# EPICS substitutions: iocBoot/ioczzz/zedLOreg6.substitutions
# base address 0x43c50000
file "$(TOP)/zzzApp/Db/zedLOreg.template"
{
pattern
{P,R,C,N, SCAN}
{zzz:,reg6_,6,0,8}
{zzz:,reg6_,6,1,8}
{zzz:,reg6_,6,2,8}
{zzz:,reg6_,6,3,8}
{zzz:,reg6_,6,4,8}
{zzz:,reg6_,6,5,8}
{zzz:,reg6_,6,6,8}
{zzz:,reg6_,6,7,8}
{zzz:,reg6_,6,8,8}
{zzz:,reg6_,6,9,8}
{zzz:,reg6_,6,10,8}
{zzz:,reg6_,6,11,8}
{zzz:,reg6_,6,12,8}
{zzz:,reg6_,6,13,8}
{zzz:,reg6_,6,14,8}
{zzz:,reg6_,6,15,8}
{zzz:,reg6_,6,16,8}
{zzz:,reg6_,6,17,8}
{zzz:,reg6_,6,18,8}
{zzz:,reg6_,6,19,8}
{zzz:,reg6_,6,20,8}
{zzz:,reg6_,6,21,8}
{zzz:,reg6_,6,22,8}
{zzz:,reg6_,6,23,8}
{zzz:,reg6_,6,24,8}
{zzz:,reg6_,6,25,8}
{zzz:,reg6_,6,26,8}
{zzz:,reg6_,6,27,8}
{zzz:,reg6_,6,28,8}
{zzz:,reg6_,6,29,8}

{zzz:,reg6_,6,30,8}
{zzz:,reg6_,6,31,8}
{zzz:,reg6_,6,32,8}
{zzz:,reg6_,6,33,8}
{zzz:,reg6_,6,34,8}
{zzz:,reg6_,6,35,8}
{zzz:,reg6_,6,36,8}
{zzz:,reg6_,6,37,8}
{zzz:,reg6_,6,38,8}
{zzz:,reg6_,6,39,8}

{zzz:,reg6_,6,40,8}
{zzz:,reg6_,6,41,8}
{zzz:,reg6_,6,42,8}
{zzz:,reg6_,6,43,8}
{zzz:,reg6_,6,44,8}
{zzz:,reg6_,6,45,8}
{zzz:,reg6_,6,46,8}
{zzz:,reg6_,6,47,8}
{zzz:,reg6_,6,48,8}
{zzz:,reg6_,6,49,8}

{zzz:,reg6_,6,50,8}
{zzz:,reg6_,6,51,8}
{zzz:,reg6_,6,52,8}
{zzz:,reg6_,6,53,8}
{zzz:,reg6_,6,54,8}
{zzz:,reg6_,6,55,8}
{zzz:,reg6_,6,56,8}
{zzz:,reg6_,6,57,8}
{zzz:,reg6_,6,58,8}
{zzz:,reg6_,6,59,8}

{zzz:,reg6_,6,60,8}
{zzz:,reg6_,6,61,8}
{zzz:,reg6_,6,62,8}
{zzz:,reg6_,6,63,8}
{zzz:,reg6_,6,64,8}
{zzz:,reg6_,6,65,8}
{zzz:,reg6_,6,66,8}
{zzz:,reg6_,6,67,8}
{zzz:,reg6_,6,68,8}
{zzz:,reg6_,6,69,8}

{zzz:,reg6_,6,70,8}
{zzz:,reg6_,6,71,8}
{zzz:,reg6_,6,72,8}
{zzz:,reg6_,6,73,8}
{zzz:,reg6_,6,74,8}
{zzz:,reg6_,6,75,8}
{zzz:,reg6_,6,76,8}
{zzz:,reg6_,6,77,8}
{zzz:,reg6_,6,78,8}
{zzz:,reg6_,6,79,8}

{zzz:,reg6_,6,80,8}
{zzz:,reg6_,6,81,8}
{zzz:,reg6_,6,82,8}
{zzz:,reg6_,6,83,8}
{zzz:,reg6_,6,84,8}
{zzz:,reg6_,6,85,8}
{zzz:,reg6_,6,86,8}
{zzz:,reg6_,6,87,8}
{zzz:,reg6_,6,88,8}
{zzz:,reg6_,6,89,8}

{zzz:,reg6_,6,90,8}
{zzz:,reg6_,6,91,8}
{zzz:,reg6_,6,92,8}
{zzz:,reg6_,6,93,8}
{zzz:,reg6_,6,94,8}
{zzz:,reg6_,6,95,8}
{zzz:,reg6_,6,96,8}
{zzz:,reg6_,6,97,8}
{zzz:,reg6_,6,98,8}
{zzz:,reg6_,6,99,8}

{zzz:,reg6_,6,100,8}
{zzz:,reg6_,6,101,8}
{zzz:,reg6_,6,102,8}
{zzz:,reg6_,6,103,8}
{zzz:,reg6_,6,104,8}
{zzz:,reg6_,6,105,8}
{zzz:,reg6_,6,106,8}
{zzz:,reg6_,6,107,8}
{zzz:,reg6_,6,108,8}
{zzz:,reg6_,6,109,8}

{zzz:,reg6_,6,110,8}
{zzz:,reg6_,6,111,8}
{zzz:,reg6_,6,112,8}
{zzz:,reg6_,6,113,8}
{zzz:,reg6_,6,114,8}
{zzz:,reg6_,6,115,8}
{zzz:,reg6_,6,116,8}
{zzz:,reg6_,6,117,8}
{zzz:,reg6_,6,118,8}
{zzz:,reg6_,6,119,8}

{zzz:,reg6_,6,120,8}
{zzz:,reg6_,6,121,8}
{zzz:,reg6_,6,122,8}
{zzz:,reg6_,6,123,8}
{zzz:,reg6_,6,124,8}
{zzz:,reg6_,6,125,8}
{zzz:,reg6_,6,126,8}
{zzz:,reg6_,6,127,8}
{zzz:,reg6_,6,128,8}
{zzz:,reg6_,6,129,8}

{zzz:,reg6_,6,130,8}
{zzz:,reg6_,6,131,8}
{zzz:,reg6_,6,132,8}
{zzz:,reg6_,6,133,8}
{zzz:,reg6_,6,134,8}
{zzz:,reg6_,6,135,8}
{zzz:,reg6_,6,136,8}
{zzz:,reg6_,6,137,8}
{zzz:,reg6_,6,138,8}
{zzz:,reg6_,6,139,8}

{zzz:,reg6_,6,140,8}
{zzz:,reg6_,6,141,8}
{zzz:,reg6_,6,142,8}
{zzz:,reg6_,6,143,8}
{zzz:,reg6_,6,144,8}
{zzz:,reg6_,6,145,8}
{zzz:,reg6_,6,146,8}
{zzz:,reg6_,6,147,8}
{zzz:,reg6_,6,148,8}
{zzz:,reg6_,6,149,8}

{zzz:,reg6_,6,150,8}
{zzz:,reg6_,6,151,8}
{zzz:,reg6_,6,152,0}
{zzz:,reg6_,6,153,0}
{zzz:,reg6_,6,154,0}
{zzz:,reg6_,6,155,0}
{zzz:,reg6_,6,156,0}
{zzz:,reg6_,6,157,0}
{zzz:,reg6_,6,158,0}
{zzz:,reg6_,6,159,0}
}
